// TwinCAT 3 PLC project PLC
// ProgramVersion: 3.1.4024.0
// libraries:
//   Tc2_Standard, * (Beckhoff Automation GmbH)
//   Tc2_System, * (Beckhoff Automation GmbH)
//   Tc3_Module, * (Beckhoff Automation GmbH)
//   VisuSymbols,3.5.10.0,System
// project tree:
//   / Gestore di visualizzazione.TcVMO (not stored), GlobalTextList.TcGTLO, PlcTask.TcTTO
//   GVLs/ GVL.TcGVL
//   POUs/ LD_Logic.TcPOU, MAIN.TcPOU
//   VISUs/ Visualization.TcVIS
// real-time tasks:
//   TASK PlcTask: cycle T#10ms, priority 20, ADS port 350

CONFIGURATION PLC
    RESOURCE PLC ON TwinCAT3
        TASK PlcTask(INTERVAL := T#10ms, PRIORITY := 20);
        PROGRAM MAIN WITH PlcTask : MAIN;
    END_RESOURCE
END_CONFIGURATION

// ---- GVLs/GVL.TcGVL
{attribute 'qualified_only'}
VAR_GLOBAL
	MachineIsActive: BOOL;
	MachineIsRunning : BOOL;
	Emergency: BOOL;
	PBStart : BOOL;
	PBStop : BOOL;
	PBEmergency: BOOL;
END_VAR

// ---- POUs/MAIN.TcPOU
PROGRAM MAIN
VAR
END_VAR

LD_Logic();

END_PROGRAM

// ---- POUs/LD_Logic.TcPOU
PROGRAM LD_Logic
VAR
END_VAR

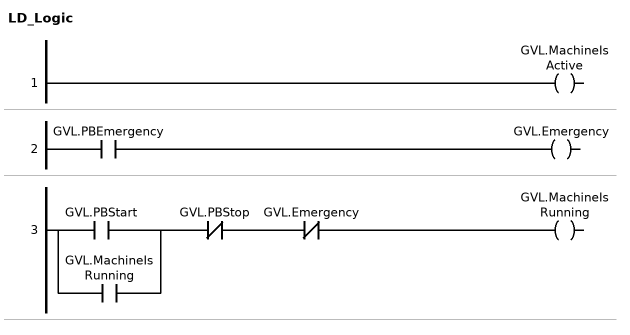
// NETWORK 1
GVL.MachineIsActive := TRUE;

// NETWORK 2
GVL.Emergency := GVL.PBEmergency;

// NETWORK 3
GVL.MachineIsRunning := (GVL.PBStart OR GVL.MachineIsRunning) AND NOT GVL.PBStop AND NOT GVL.Emergency;

END_PROGRAM

// ---- GlobalTextList.TcGTLO
TEXTLIST GlobalTextList
  849 = 'Emergenza'
  284 = 'Start'
  796 = 'Stop'
  606 = 'Testo'
END_TEXTLIST

// ---- VISUs/Visualization.TcVIS
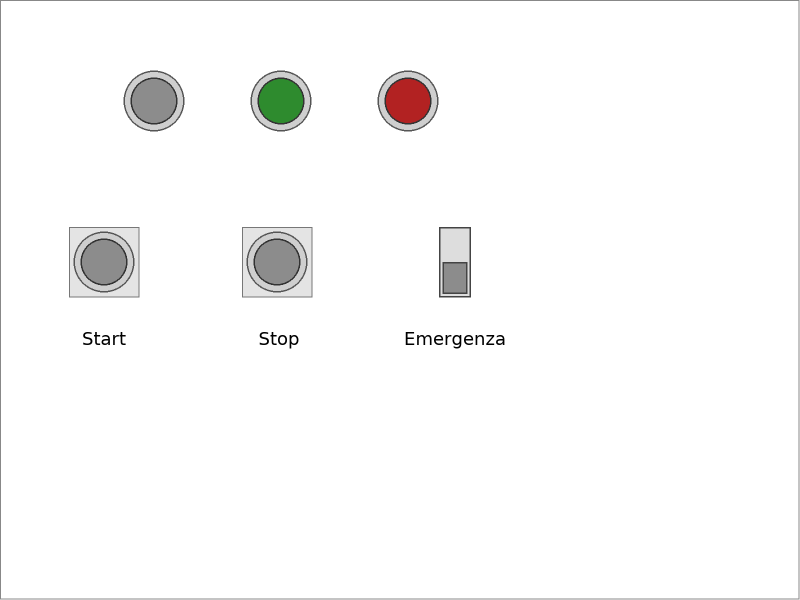
VISUALIZATION Visualization  // 800x600
    Label (29,324 150x30), "Start"
    Lamp1 (119,66 70x70), variable: GVL.MachineIsActive, style: Lamp-Lamp1-Gray
    Lamp1 (246,66 70x70), variable: GVL.MachineIsRunning, style: Lamp-Lamp1-Green
    Lamp1 (373,66 70x70), variable: GVL.Emergency, style: Lamp-Lamp1-Red
    PushSwitch (69,227 70x70), variable: GVL.PBStart, behaviour: TAP, style: Switch-PushSwitch-Gray
    Label (204,324 150x30), "Stop"
    PushSwitch (242,227 70x70), variable: GVL.PBStop, behaviour: TAP, style: Switch-PushSwitch-Gray
    DipSwitch (420,227 70x70), variable: GVL.PBEmergency, behaviour: TOGGLE, style: Switch-DipSwitch-Gray
    Label (380,324 150x30), "Emergenza"
END_VISUALIZATION
